FUNCTION_BLOCK ZephyrIO (* Template for Modular IO with boards running Zephyr OS *)
  (* Standard: 61499-2; Description: Copyright (c) 2024 Dirk Kaar This program and the accompanying materials are made available under the terms of the Eclipse Public License 2.0 which is available at https://www.eclipse.org/legal/epl-2.0/ SPDX-License-Identifier: EPL-2.0 Contributors: Dirk Kaar *)
  (* Version 1.0, 2024-01-12, Dirk Kaar *)
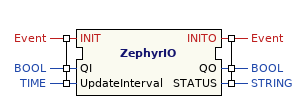
  EVENT_INPUT
    INIT WITH QI, UpdateInterval; (* Service Initialization *)
  END_EVENT
  EVENT_OUTPUT
    INITO WITH QO, STATUS; (* Initialization Confirm *)
  END_EVENT
  VAR_INPUT
    QI : BOOL; (* Event Input Qualifier *)
    UpdateInterval : TIME := T#40ms; (* Update interval *)
  END_VAR
  VAR_OUTPUT
    QO : BOOL; (* Event Output Qualifier *)
    STATUS : STRING; (* Service Status *)
  END_VAR
  (* Service APPLICATION/RESOURCE: Template for Modular IO with boards running Zephyr OS *)
END_FUNCTION_BLOCK
